FUNCTION_BLOCK FB_Module
VAR_INPUT
END_VAR
VAR_OUTPUT
END_VAR
VAR
END_VAR

END_FUNCTION_BLOCK

(* stored: Version 1.1.0.1, ProductVersion 3.1.4026.17
   POU FB_Module: Id {245e3b14-486a-4d3d-b47e-47bddc614d02}, SpecialFunc None *)
